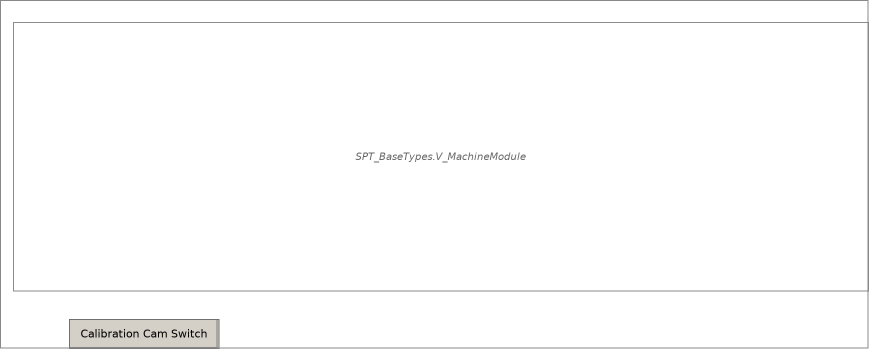
VISUALIZATION Visualization  // 869x349
    Frame (13,22 856x269)
        shows SPT_BaseTypes.V_MachineModule(HMI := MAIN.Machine.PackMLBaseModule_HMI)
    Button (69,319 150x30), "Calibration Cam Switch"
        toggle MAIN.Machine.CalibrationCam._CalibrationCam
END_VISUALIZATION

(* stored: Version 1.1.0.1, ProductVersion 3.1.4026.12
   Visu Visualization: Id {5be74494-91dd-4b66-826f-b48c7fe0c03b} *)
